// TIA Portal project "Greifen_und_Sortieren_0" (V20)

(* hardware
DEVICE "S7-1500/ET200MP-Station_1"  S7-1500 station
   slot 0: "Profilschiene_0"  Rack  6ES7 590-1***0-0AA0
   slot 1: "PLC_1"  CPU 1513-1 PN  6ES7 513-1AM03-0AB0  V4.0
      slot 3: "CPU-Display_1"  6ES7591-1AA00-0AA0
      slot 32768: "PROFINET-Schnittstelle_1"  X1
         slot 32769: "Port_1"  X1 P1
         slot 32770: "Port_2"  X1 P2
      slot 34817: "Virtual CP interface port_1"  Virtual CP interface port  Virtual CP interface port FW V4.0
   slot 2: "DI 16x24VDC BA_1"  DI 16x24VDC BA  6ES7 521-1BH10-0AA0  V1.1
   slot 3: "DQ 16x24VDC/0.5A ST_1"  DQ 16x24VDC/0.5A ST  6ES7 522-1BH00-0AB0  V2.0
   slot 4: "AI 8xU/I/R/RTD BA_1"  AI 8xU/I/R/RTD BA  6ES7 531-7QF00-0AB0  V1.0
   slot 5: "AQ 8xU/I HS_1"  AQ 8xU/I HS  6ES7 532-5HF00-0AB0  V2.2
   slot 6: "AI 8xU/I/R/RTD BA_2"  AI 8xU/I/R/RTD BA  6ES7 531-7QF00-0AB0  V1.0
   slot 7: "AQ 8xU/I HS_2"  AQ 8xU/I HS  6ES7 532-5HF00-0AB0  V2.2
*)

// ===== PLC "PLC_1"  CPU 1513-1 PN =====

VAR_GLOBAL   // PLC tag table "Standard-Variablentabelle"
   "PlcLabConnectIn01" AT %ID32760 : DWord;
   "PlcLabConnectIn02" AT %ID32764 : DWord;
   "PlcLabConnectOut01" AT %QD32760 : DWord;
   "PlcLabConnectOut02" AT %QD32764 : DWord;
   "NotAus_aktiv" AT %M1.0 : Bool;
   "Clock_Byte" AT %MB0 : Byte;
   "Clock_10Hz" AT %M0.0 : Bool;
   "Clock_5Hz" AT %M0.1 : Bool;
   "Clock_2.5Hz" AT %M0.2 : Bool;
   "Clock_2Hz" AT %M0.3 : Bool;
   "Clock_1.25Hz" AT %M0.4 : Bool;
   "Clock_1Hz" AT %M0.5 : Bool;
   "Clock_0.625Hz" AT %M0.6 : Bool;
   "Clock_0.5Hz" AT %M0.7 : Bool;
   "Anlage_aktiv" AT %M1.1 : Bool;
   "Ein_Paket_erkannt" AT %M1.2 : Bool;
   "Prozess_beendet" AT %M2.7 : Bool;
   "Paket_im_Auslauf" AT %M1.3 : Bool;
   "Greifer_runter" AT %M2.0 : Bool;
   "Greifen" AT %M2.1 : Bool;
   "Greifer_hoch" AT %M2.2 : Bool;
   "Loslassen" AT %M2.3 : Bool;
   "X_ansteuern" AT %M2.4 : Bool;
   "Z_ansteuern" AT %M2.5 : Bool;
   "Greifer_einfahren" AT %M2.6 : Bool;
   "Z_bewegt" AT %M3.0 : Bool;
   "X_bewegt" AT %M3.1 : Bool;
   "Zaehler_zurueck" AT %M3.2 : Bool;
   "Aus_Paket_erkannt" AT %M1.4 : Bool;
   "Aus_Band_fertig" AT %M1.5 : Bool;
   "Prozess_starten" AT %M3.3 : Bool;
END_VAR

VAR_GLOBAL   // PLC tag table "Eingaenge"
   "S1" AT %I0.0 : Bool;   // Not-Aus
   "S2" AT %I0.1 : Bool;   // Betriebsschalter
   "S3" AT %I0.2 : Bool;   // Starttaster
   "S4" AT %I0.3 : Bool;   // Stopptaster
   "S5" AT %I0.4 : Bool;   // Resettaster
   "1b1" AT %I0.5 : Bool;   // Einlaufband Sensor
   "1b2" AT %I0.6 : Bool;   // Auslaufband Sensor
   "2b1" AT %I1.0 : Bool;   // Greifer Z-Achse Bewegung
   "2b2" AT %I1.1 : Bool;   // Greifer X-Achse Bewegung
   "2b3" AT %I1.2 : Bool;   // Greifer greft
END_VAR

VAR_GLOBAL   // PLC tag table "Ausgaenge"
   "H1" AT %Q0.2 : Bool;   // Startleuchte
   "H2" AT %Q0.3 : Bool;   // Stoppleuchte
   "H3" AT %Q0.4 : Bool;   // Resetleuchte
   "M1" AT %Q0.5 : Bool;   // Einlaufband
   "M2" AT %Q0.6 : Bool;   // Auslaufband
   "M3" AT %Q1.0 : Bool;   // Greifer Z-Achse bewegen
   "M4" AT %Q1.1 : Bool;   // Greifer X-Achse bewegen
   "M5" AT %Q1.2 : Bool;   // Greifer greifen
   "D1" AT %QD30 : DInt;   // Zähler
END_VAR

// folder: System blocks/Program resources

DATA_BLOCK "IEC_Timer_0_DB"   // DB1
{ S7_Optimized_Access := 'TRUE' }
AUTHOR : Simatic
FAMILY : IEC
NAME : IEC_TMR
VERSION : 1.0
// stored: InstanceOfName IEC_TIMER
"IEC_TIMER"
BEGIN
END_DATA_BLOCK

DATA_BLOCK "IEC_Counter_0_DB"   // DB2
{ S7_Optimized_Access := 'TRUE' }
AUTHOR : Simatic
FAMILY : IEC
NAME : CNTR
VERSION : 1.0
// stored: InstanceOfName IEC_COUNTER
"IEC_COUNTER"
BEGIN
END_DATA_BLOCK

DATA_BLOCK "IEC_Counter_0_DB_1"   // DB3
{ S7_Optimized_Access := 'TRUE' }
AUTHOR : Simatic
FAMILY : IEC
NAME : CNTR
VERSION : 1.0
// stored: InstanceOfName IEC_COUNTER
"IEC_COUNTER"
BEGIN
END_DATA_BLOCK

// folder: (top level)

FUNCTION "Greifersteuerung" : Void   // FC1, FBD
{ S7_Optimized_Access := 'TRUE' }
VERSION : 0.1
   VAR_TEMP
      Z_Zaehler : Int;
      Mod_Z_Zaehler : Int;
   END_VAR
   VAR_TEMP   // added for the SCL form of the ladder/FBD networks
      _w1 : Bool;
      _w2 : Bool;
   END_VAR
BEGIN

REGION Network 1: Anlagensteuerung
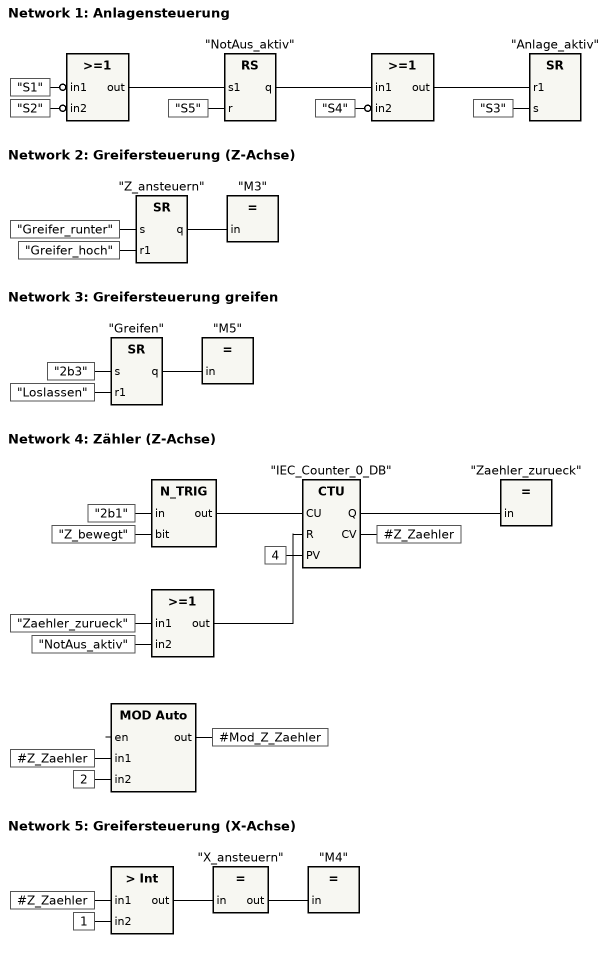
   IF "S5" THEN
       "NotAus_aktiv" := FALSE;   // RS flip-flop
   END_IF;
   IF NOT "S1" OR NOT "S2" THEN "NotAus_aktiv" := TRUE; END_IF;
   IF "S3" THEN
       "Anlage_aktiv" := TRUE;   // SR flip-flop
   END_IF;
   IF "NotAus_aktiv" OR NOT "S4" THEN "Anlage_aktiv" := FALSE; END_IF;
END_REGION

REGION Network 2: Greifersteuerung (Z-Achse)
   IF "Greifer_runter" THEN
       "Z_ansteuern" := TRUE;   // SR flip-flop
   END_IF;
   IF "Greifer_hoch" THEN "Z_ansteuern" := FALSE; END_IF;
   "M3" := "Z_ansteuern";
END_REGION

REGION Network 3: Greifersteuerung greifen
   IF "2b3" THEN
       "Greifen" := TRUE;   // SR flip-flop
   END_IF;
   IF "Loslassen" THEN "Greifen" := FALSE; END_IF;
   "M5" := "Greifen";
END_REGION

REGION Network 4: Zähler (Z-Achse)
   #_w1 := NOT "2b1" AND "Z_bewegt";   // falling edge
   "Z_bewegt" := "2b1";
   "IEC_Counter_0_DB".CTU(CU := #_w1, R := "Zaehler_zurueck" OR "NotAus_aktiv", PV := 4, CV => #Z_Zaehler);
   "Zaehler_zurueck" := "IEC_Counter_0_DB".Q;
   #Mod_Z_Zaehler := #Z_Zaehler MOD 2;
END_REGION

REGION Network 5: Greifersteuerung (X-Achse)
   "X_ansteuern" := #Z_Zaehler > 1;
   "M4" := "X_ansteuern";
END_REGION

REGION Network 6: Greiferprozessschritte
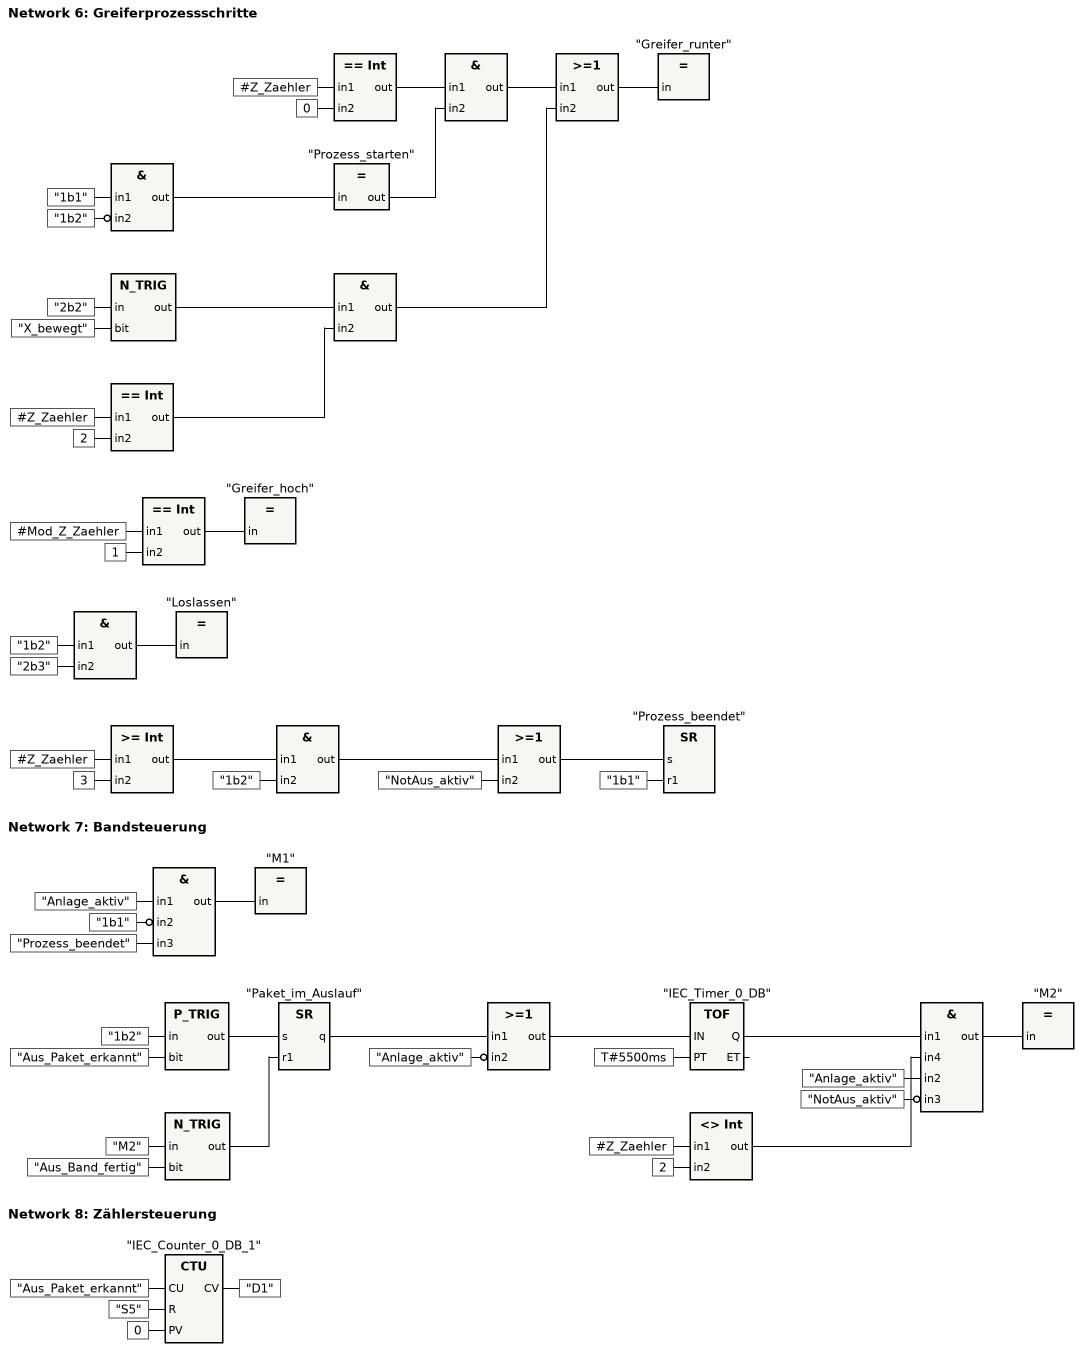
   "Prozess_starten" := "1b1" AND NOT "1b2";
   #_w1 := NOT "2b2" AND "X_bewegt";   // falling edge
   "X_bewegt" := "2b2";
   "Greifer_runter" := ((#Z_Zaehler = 0) AND "Prozess_starten") OR (#_w1 AND (#Z_Zaehler = 2));
   "Greifer_hoch" := #Mod_Z_Zaehler = 1;
   "Loslassen" := "1b2" AND "2b3";
   IF ((#Z_Zaehler >= 3) AND "1b2") OR "NotAus_aktiv" THEN
       "Prozess_beendet" := TRUE;   // SR flip-flop
   END_IF;
   IF "1b1" THEN "Prozess_beendet" := FALSE; END_IF;
END_REGION

REGION Network 7: Bandsteuerung
   "M1" := "Anlage_aktiv" AND NOT "1b1" AND "Prozess_beendet";
   #_w1 := "1b2" AND NOT "Aus_Paket_erkannt";   // rising edge
   "Aus_Paket_erkannt" := "1b2";
   #_w2 := NOT "M2" AND "Aus_Band_fertig";   // falling edge
   "Aus_Band_fertig" := "M2";
   IF #_w1 THEN
       "Paket_im_Auslauf" := TRUE;   // SR flip-flop
   END_IF;
   IF #_w2 THEN "Paket_im_Auslauf" := FALSE; END_IF;
   "IEC_Timer_0_DB".TOF(IN := "Paket_im_Auslauf" OR NOT "Anlage_aktiv", PT := T#5500ms);
   "M2" := "IEC_Timer_0_DB".Q AND (#Z_Zaehler <> 2) AND "Anlage_aktiv" AND NOT "NotAus_aktiv";
END_REGION

REGION Network 8: Zählersteuerung
   "IEC_Counter_0_DB_1".CTU(CU := "Aus_Paket_erkannt", R := "S5", PV := 0, CV => "D1");
END_REGION

REGION Network 9: Beleuchtungssteuerung
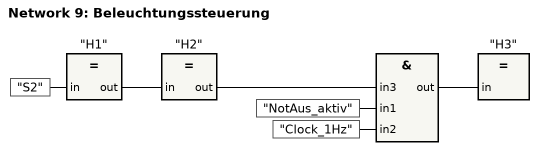
   "H1" := "S2";
   "H2" := "S2";
   "H3" := "S2" AND "NotAus_aktiv" AND "Clock_1Hz";
END_REGION
END_FUNCTION

ORGANIZATION_BLOCK "Main"   // OB1, FBD, ProgramCycle
TITLE = "Main Program Sweep (Cycle)"
{ S7_Optimized_Access := 'TRUE' }
VERSION : 0.1
   VAR_INPUT
      Initial_Call : Bool;   // Initial call of this OB
      Remanence : Bool;   // =True, if remanent data are available
   END_VAR
BEGIN

REGION Network 1
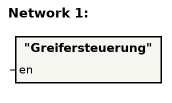
   "Greifersteuerung"();
END_REGION
END_ORGANIZATION_BLOCK